PROGRAM MAIN
VAR
	nastro	:	FB_MSF();
END_VAR

nastro(
	start:= IO.start, 
	stop:= IO.stop, 
	emg:= IO.emg, 
	ack:= IO.ack, 
	fc1:= IO.fc1, 
	fc2:= IO.fc2, 
	H1=> IO.H1, 
	HEMG=> IO.HEMG, 
	M=> IO.M, 
	libero=> IO.libero);

END_PROGRAM

(* stored: Version 1.1.0.1, ProductVersion 3.1.4024.12
   POU MAIN: Id {61fcc61d-2ea2-427b-827c-c7a65c42e900}, SpecialFunc None *)
